FUNCTION_BLOCK StartMovementsTask  EXTENDS TcoAbbRoboticsTask
VAR
     _moveParams:TcoAbstractions.TcoRoboticsMovementsParams;
	 
	 
END_VAR


IF Execute() THEN
	IF _progress = 0 THEN
		IF NOT __ISVALIDREF(inoControl) THEN
			_varInfo :=__VARINFO(inoControl);
			Messenger.Programming(_sb.Clear().Append('<#Invalid reference: #>').Append(_varInfo.Symbol).ToString()).Pin();
		ELSIF NOT __ISVALIDREF(inoConfig) THEN                                                  
			_varInfo :=__VARINFO(inoConfig);                                                    
			Messenger.Programming(_sb.Clear().Append('<#Invalid reference: #>').Append(_varInfo.Symbol).ToString()).Pin();
		ELSIF NOT __ISVALIDREF(inoStatus) THEN                                                  
			_varInfo :=__VARINFO(inoStatus);                                                    
			Messenger.Programming(_sb.Clear().Append('<#Invalid reference: #>').Append(_varInfo.Symbol).ToString()).Pin();
			ELSE
			_progress := _progress + 1;
		END_IF

	END_IF
	
	IF _progress = 1 THEN
		
		_varInfo :=__VARINFO( inoStatus.State.CycleOn);                                                
		THIS^.Messenger.OnCondition(_infoTimer.Q AND NOT inoStatus.State.CycleOn).Warning(_sb.Clear().Append('<#Waiting for program running signal! #>').Append(_varInfo.Symbol).ToString());
		
		_varInfo :=__VARINFO( inoStatus.State.MotorOnState);                                                
		THIS^.Messenger.OnCondition(_infoTimer.Q AND NOT inoStatus.State.MotorOnState).Warning(_sb.Clear().Append('<#Waiting for motors are On! #>').Append(_varInfo.Symbol).ToString());	
		
		_varInfo :=__VARINFO( inoStatus.State.Error);                                                
		THIS^.Messenger.OnCondition(_infoTimer.Q AND inoStatus.State.Error).Warning(_sb.Clear().Append('<#Waiting for system is without errors! #>').Append(_varInfo.Symbol).ToString());
		
		IF inoStatus.State.CycleOn AND inoStatus.State.MotorOnState AND NOT inoStatus.State.Error THEN 
			_progress := _progress + 1;
		END_IF

	END_IF;
	
	
	IF _progress = 2 THEN
		inoControl.GlobalSpeed := _moveParams.GlobalSpeed;
		inoControl.ToolNo := _moveParams.ToolNo;
		inoControl.WorkobjectNo := _moveParams.WorkobjectNo;
		inoControl.PointNo := _moveParams.PointNo;
		inoControl.UserSpecSpeed1 := _moveParams.UserSpecSpeed1;
		inoControl.UserSpecSpeed2 := _moveParams.UserSpecSpeed2;
		inoControl.Coordinates := _moveParams.Coordinates; 		
	
		inoControl.ActionNo := 254;
		IF inoControl.ActionNo = inoStatus.State.ActionNo THEN
			
			_progress:=_progress + 1;
		END_IF
	END_IF;	
	IF _progress = 3 THEN
		IF 	inoStatus.State.GlobalSpeed = _moveParams.GlobalSpeed AND
			inoStatus.State.ToolNo = _moveParams.ToolNo AND
			inoStatus.State.WorkobjectNo = _moveParams.WorkobjectNo AND
			inoStatus.State.PointNo = _moveParams.PointNo AND
			inoStatus.State.UserSpecSpeed1 = _moveParams.UserSpecSpeed1 AND
			inoStatus.State.UserSpecSpeed2 =_moveParams.UserSpecSpeed2 AND
			TcoAbstractions.CoordinatesAreEqual(inoStatus.State.Coordinates,_moveParams.Coordinates,0.01,0.01,0.01,0.01,0.01,0.01) THEN
			inoControl.ActionNo := 255;
			_progress:=_progress + 1;
		END_IF
	END_IF;	
	
	IF _progress = 4 THEN
		IF inoControl.ActionNo = inoStatus.State.ActionNo THEN
			_progress:=_progress + 1;
		END_IF
	END_IF;	
	
	
	
	IF _progress = 5 THEN
	
		Messenger.Info(CONCAT('<#Moving to position ID#>: ', INT_TO_STRING(_moveParams.ActionNo)));
		inoControl.ActionNo := _moveParams.ActionNo;
		IF inoControl.ActionNo = inoStatus.State.ActionNo THEN
			inoControl.ActionNo :=255;
				_progress := _progress + 1;
		END_IF
	END_IF;		
			
	IF _progress = 6 THEN
		IF inoControl.ActionNo = inoStatus.State.ActionNo THEN
			 DoneWhen(TRUE);
		END_IF
	END_IF;		

   CallTimers(TRUE);
	
	THIS^.ThrowWhen(_errorTimer.Q OR inoStatus.State.Error);
END_IF

IF  THIS^.Error AND NOT _errorMessage.Pinned THEN
	THIS^.Restore();
END_IF

METHOD PUBLIC FB_init : BOOL
VAR_INPUT
    bInitRetains : BOOL; // if TRUE, the retain variables are initialized (warm start / cold start)
    bInCopyCode : BOOL; // if TRUE, the instance afterwards gets moved into the copy code (online change)
  	ParentObject : ITcoObject;	
END_VAR
END_METHOD

METHOD INTERNAL InvokeWithParams : ITcoTaskStatus
VAR_INPUT
    inMoveParams:TcoAbstractions.TcoRoboticsMovementsParams;
END_VAR
_moveParams:=inMoveParams;
InvokeWithParams := THIS^.Invoke();
END_METHOD

(*~
	<docu>
		<summary>
			Executes when task is aborted.
		</summary>			
	</docu>	
~*)
METHOD PROTECTED OnAbort
IF  __ISVALIDREF(inoStatus) THEN   THIS^.inoStatus.ActionDescription := '<#Start movements was aborted, while not yet completed!#>';END_IF; 
inoControl.SoftStop := TRUE;
inoControl.QuickStop := FALSE;
END_METHOD

(*~
	<docu>
		<summary>
			Executes when task reaches the ```Done``` state .
		</summary>			
	</docu>	
~*)
METHOD PROTECTED OnDone
IF  __ISVALIDREF(inoStatus) THEN   THIS^.inoStatus.ActionDescription := '<#Start movements finished successfully.#>'; END_IF;
_progress:=0;
END_METHOD

(*~
	<docu>
		<summary>
			Executes when task reaches the ```Error``` state.
		
		</summary>			
	</docu>	
~*)
METHOD PROTECTED OnError
VAR
	description: STRING;
END_VAR
description := '<#Start movements finished with error.#>'; 
IF  __ISVALIDREF(inoStatus) THEN   THIS^.inoStatus.ActionDescription := description; END_IF;
THIS^._errorMessage.Error(_sb.Clear().Append(description).Append(' To restore acknowledge this alarm.').ToString()).Pin();
END_METHOD

METHOD PROTECTED OnStart
IF  __ISVALIDREF(inoStatus) THEN   THIS^.inoStatus.ActionDescription := '<#Start movements stared.#>'; END_IF;
CallTimers(FALSE);
inoControl.QuickStop:=FALSE;
inoControl.SoftStop:=FALSE;
END_METHOD

(*~
	<docu>
		<summary>
			Restores this instance to the Ready state. Can be called explicitly or from within one of the restore mechanisms.
			<para>
				See also <see cref="PlcDocu.TcoCore.TcoTask.AutoRestorable()"/>
			</para>
		</summary>			
	</docu>	
~*)
METHOD Restore : ITcoRestorable
SUPER^.Restore();
END_METHOD

END_FUNCTION_BLOCK

(* stored: Version 1.1.0.1, ProductVersion 3.1.4024.12
   POU StartMovementsTask: Id {f3921a87-3dfe-0477-2012-ac3d2b31e7d2}, SpecialFunc None
   Method FB_init: Id {7bb61c04-c516-0af1-30da-1fe46e27df62}
   Method InvokeWithParams: Id {0b0d78d7-fe60-0ca4-022c-1c877dbbe624}
   Method OnAbort: Id {41060f6f-931e-0bf0-02ea-bf599a1c82eb}
   Method OnDone: Id {eae494ac-5e3e-0708-28d6-d356d06c2c34}
   Method OnError: Id {9e3a3e6b-cd53-0a32-2a83-e8852c3ea144}
   Method OnStart: Id {ae09c0fb-a1ed-0ee7-369e-7e5f9c72c591}
   Method Restore: Id {3a02f0ca-89c2-0708-2606-32ca64d615ba} *)
